# EPICS substitutions: iocs/MC05/db/SAI_DigitalChannels.substitutions
file /opt/epics/modules/SAI/db/SAI_DigitalChannels.template {
pattern {	P,		R,		SCAN, 		ASYNPORT}
        { 	"XF:06BM-OP",		"{MC:05}",	"1 second",	"pmac"}
}

#EOF
